// TIA Portal project "Grundkurs Aufgabe 3 NEU" (V15.1)
// Vorlageprojekt für das Buch mit Zielsystem S7-1200

(* hardware
DEVICE "S7-1200-Station_1"  S7-1200 Station
   slot 0: "Baugruppenträger_0"  Rack  V1.0
   slot 1: "SPS"  CPU 1212C AC/DC/Rly  6ES7 212-1BE40-0XB0  V4.2
*)

// ===== PLC "SPS"  CPU 1212C AC/DC/Rly =====

VAR_GLOBAL   // PLC tag table "Eingänge und Ausgänge"
   "Taster_Start" AT %E0.0 : Bool;   // Taster "Start" Bedienpult (Schließer)
   "NotAus" AT %E0.2 : Bool;   // NotAus Bedienpult (Öffner)
   "Lichttaster_Auslauf" AT %E0.4 : Bool;   // Lichttaster im Auslauf des Förderbandes (Schließer)
   "Motor_Foerderband" AT %A0.2 : Bool;   // Motor Förderband vorwärts
   "Rundumleuchte" AT %A0.3 : Bool;   // Rundumleuchte über Bedienpult
   "Taster_Stop" AT %E0.1 : Bool;   // Taster "Stop" Bedienpult (Öffner)
   "Leuchte_Start" AT %A0.0 : Bool;   // Leuchte "Start" Bedienpult
   "Leuchte_Stop" AT %A0.1 : Bool;   // Leuchte "Stop" Bedienpult
   "Lichttaster_Einlauf" AT %E0.3 : Bool;   // Lichttaster im Einlauf des Förderbandes (Schließer)
END_VAR

VAR_GLOBAL   // PLC tag table "Merker"
   "Anlage_Start" AT %M1.0 : Bool;   // Anlage läuft
   "Foerderband_belegt" AT %M1.1 : Bool;   // Paket liegt auf Förderband
END_VAR

FUNCTION "Kopplung_FactoryIO_mit_PLCSIM" : Void   // FC9000, SCL
{ S7_Optimized_Access := 'TRUE' }
VERSION : 0.1
   VAR_TEMP
      rdTimeReturn : Int;
      outputTime : DTL;
      SyncVal : Byte;
      forVal : Int;
      forVal_2 : Int;
      Value : Byte;
   END_VAR
   VAR CONSTANT
      CompVal : Byte := 16#34;
      Value_01 : Byte := 16#11;
      Value_01_DW : DWord := 16#A165_D992;
      Value_02_DW : DWord := 16#58BE_4401;
   END_VAR
BEGIN

   #Value:=PEEK(area := 16#82,
        dbNumber := 0,
        byteOffset := 511);
   #Value := #Value + 1;

   POKE(area := 16#82,
        dbNumber := 0,
        byteOffset := 511,
        value := #Value);

   POKE(area:=16#81,
        dbNumber:=0,
        byteOffset:=1016,
        value:=#Value_01_DW);
   POKE(area := 16#81,
        dbNumber := 0,
        byteOffset := 1020,
        value := #Value_02_DW);

   POKE(area := 16#81,
        dbNumber := 0,
        byteOffset := 511,
        value := B#16#00);

   FOR #forVal := 0 TO 120 DO
       FOR #forVal_2:=0 TO 10 DO
           #rdTimeReturn:=RD_SYS_T(#outputTime);
           #rdTimeReturn := WR_SYS_T(#outputTime);
           #rdTimeReturn := RD_SYS_T(#outputTime);
           #rdTimeReturn := WR_SYS_T(#outputTime);
       END_FOR;
       #SyncVal:= PEEK(area := 16#81,
                      dbNumber := 0,
                      byteOffset := 511);
       IF #SyncVal = #CompVal THEN
          GOTO M_1;
       END_IF;
   END_FOR;
   RETURN;

   M_1:
   POKE(area := 16#81,
        dbNumber := 0,
        byteOffset := 511,
        value := B#16#0);
END_FUNCTION

ORGANIZATION_BLOCK "Main"   // OB1, FBD, ProgramCycle
TITLE = "Main Program Sweep (Cycle)"
{ S7_Optimized_Access := 'TRUE' }
VERSION : 0.1
   VAR_INPUT
      Initial_Call : Bool;   // Initial call of this OB
      Remanence : Bool;   // =True, if remanent data are available
   END_VAR
BEGIN

REGION Network 1: Konnektierungsbaustein für PLC-Lab / Bausteinaufruf FC9000 (Für Aufgabe nicht relevant)
   // Im Netzwerk 1 wird der Konnektierungsbaustein für PLC-Lab aufgerufen.
   // Dieser Aufruf darf nicht entfernt werden!
   // Der Baustein FC9000 organisiert den Datentransfer zwischen PLCSIM und FactoryIO.
   // Der Baustein kann als Beispielprojekt von der FactoryIO-Homepage heruntergeladen werden.
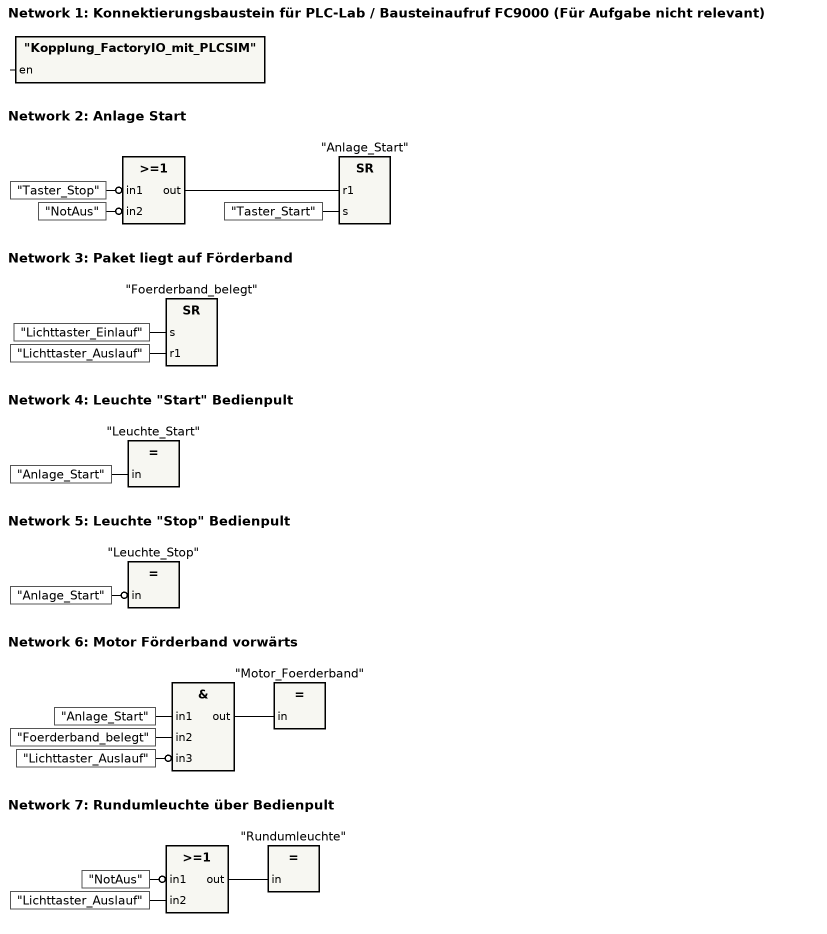
   "Kopplung_FactoryIO_mit_PLCSIM"();
END_REGION

REGION Network 2: Anlage Start
   IF "Taster_Start" THEN
       "Anlage_Start" := TRUE;   // SR flip-flop
   END_IF;
   IF NOT "Taster_Stop" OR NOT "NotAus" THEN "Anlage_Start" := FALSE; END_IF;
END_REGION

REGION Network 3: Paket liegt auf Förderband
   IF "Lichttaster_Einlauf" THEN
       "Foerderband_belegt" := TRUE;   // SR flip-flop
   END_IF;
   IF "Lichttaster_Auslauf" THEN "Foerderband_belegt" := FALSE; END_IF;
END_REGION

REGION Network 4: Leuchte "Start" Bedienpult
   "Leuchte_Start" := "Anlage_Start";
END_REGION

REGION Network 5: Leuchte "Stop" Bedienpult
   "Leuchte_Stop" := NOT "Anlage_Start";
END_REGION

REGION Network 6: Motor Förderband vorwärts
   "Motor_Foerderband" := "Anlage_Start" AND "Foerderband_belegt" AND NOT "Lichttaster_Auslauf";
END_REGION

REGION Network 7: Rundumleuchte über Bedienpult
   "Rundumleuchte" := NOT "NotAus" OR "Lichttaster_Auslauf";
END_REGION
END_ORGANIZATION_BLOCK